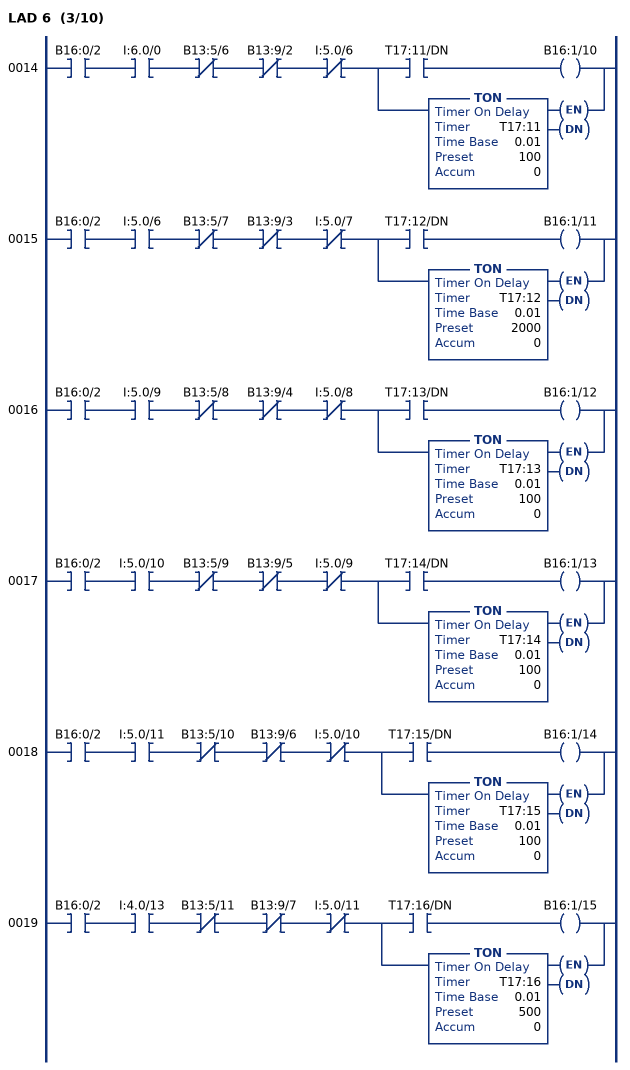
% Rung: 14 %
SOR XIC B16:0/2 XIC I:6.0/0 XIO B13:5/6 XIO B13:9/2 XIO I:5.0/6 BST XIC T17:11/DN OTE B16:1/10 NXB TON T17:11 0.01 100 0 BND EOR
% Rung: 15 %
SOR XIC B16:0/2 XIC I:5.0/6 XIO B13:5/7 XIO B13:9/3 XIO I:5.0/7 BST XIC T17:12/DN OTE B16:1/11 NXB TON T17:12 0.01 2000 0 BND EOR
% Rung: 16 %
SOR XIC B16:0/2 XIC I:5.0/9 XIO B13:5/8 XIO B13:9/4 XIO I:5.0/8 BST XIC T17:13/DN OTE B16:1/12 NXB TON T17:13 0.01 100 0 BND EOR
% Rung: 17 %
SOR XIC B16:0/2 XIC I:5.0/10 XIO B13:5/9 XIO B13:9/5 XIO I:5.0/9 BST XIC T17:14/DN OTE B16:1/13 NXB TON T17:14 0.01 100 0 BND EOR
% Rung: 18 %
SOR XIC B16:0/2 XIC I:5.0/11 XIO B13:5/10 XIO B13:9/6 XIO I:5.0/10 BST XIC T17:15/DN OTE B16:1/14 NXB TON T17:15 0.01 100 0 BND EOR
% Rung: 19 %
SOR XIC B16:0/2 XIC I:4.0/13 XIO B13:5/11 XIO B13:9/7 XIO I:5.0/11 BST XIC T17:16/DN OTE B16:1/15 NXB TON T17:16 0.01 500 0 BND EOR

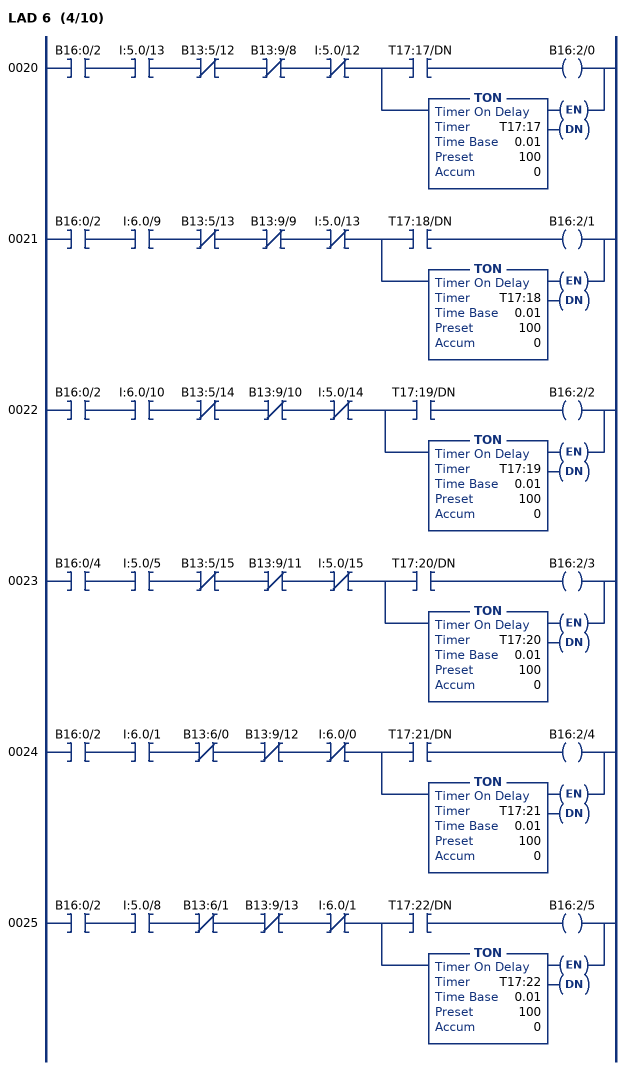
% Rung: 20 %
SOR XIC B16:0/2 XIC I:5.0/13 XIO B13:5/12 XIO B13:9/8 XIO I:5.0/12 BST XIC T17:17/DN OTE B16:2/0 NXB TON T17:17 0.01 100 0 BND EOR
% Rung: 21 %
SOR XIC B16:0/2 XIC I:6.0/9 XIO B13:5/13 XIO B13:9/9 XIO I:5.0/13 BST XIC T17:18/DN OTE B16:2/1 NXB TON T17:18 0.01 100 0 BND EOR
% Rung: 22 %
SOR XIC B16:0/2 XIC I:6.0/10 XIO B13:5/14 XIO B13:9/10 XIO I:5.0/14 BST XIC T17:19/DN OTE B16:2/2 NXB TON T17:19 0.01 100 0 BND EOR
% Rung: 23 %
SOR XIC B16:0/4 XIC I:5.0/5 XIO B13:5/15 XIO B13:9/11 XIO I:5.0/15 BST XIC T17:20/DN OTE B16:2/3 NXB TON T17:20 0.01 100 0 BND EOR
% Rung: 24 %
SOR XIC B16:0/2 XIC I:6.0/1 XIO B13:6/0 XIO B13:9/12 XIO I:6.0/0 BST XIC T17:21/DN OTE B16:2/4 NXB TON T17:21 0.01 100 0 BND EOR
% Rung: 25 %
SOR XIC B16:0/2 XIC I:5.0/8 XIO B13:6/1 XIO B13:9/13 XIO I:6.0/1 BST XIC T17:22/DN OTE B16:2/5 NXB TON T17:22 0.01 100 0 BND EOR

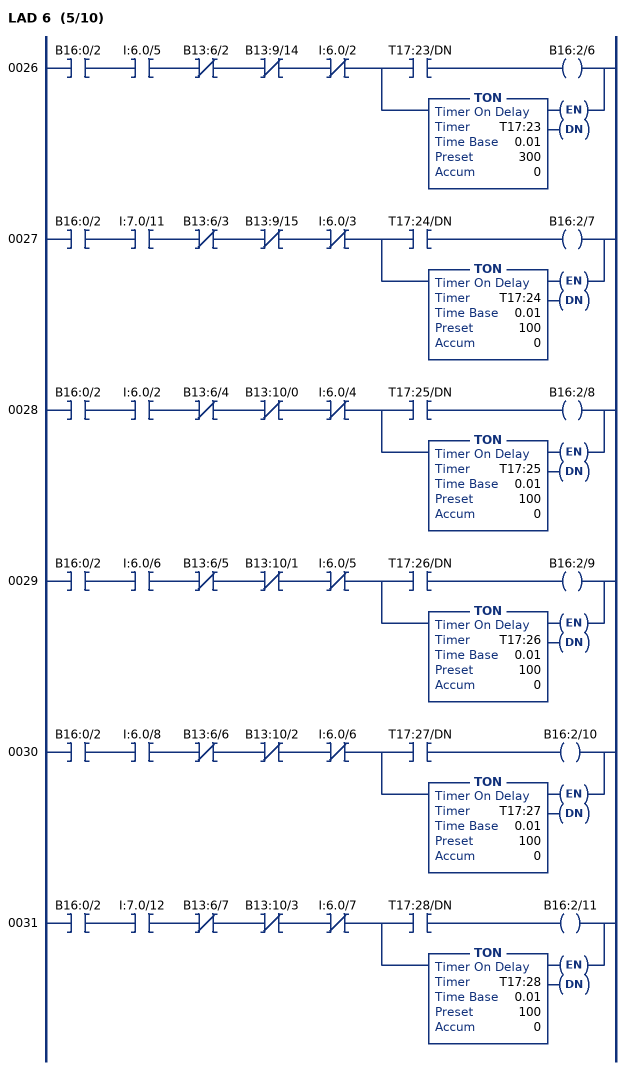
% Rung: 26 %
SOR XIC B16:0/2 XIC I:6.0/5 XIO B13:6/2 XIO B13:9/14 XIO I:6.0/2 BST XIC T17:23/DN OTE B16:2/6 NXB TON T17:23 0.01 300 0 BND EOR
% Rung: 27 %
SOR XIC B16:0/2 XIC I:7.0/11 XIO B13:6/3 XIO B13:9/15 XIO I:6.0/3 BST XIC T17:24/DN OTE B16:2/7 NXB TON T17:24 0.01 100 0 BND EOR
% Rung: 28 %
SOR XIC B16:0/2 XIC I:6.0/2 XIO B13:6/4 XIO B13:10/0 XIO I:6.0/4 BST XIC T17:25/DN OTE B16:2/8 NXB TON T17:25 0.01 100 0 BND EOR
% Rung: 29 %
SOR XIC B16:0/2 XIC I:6.0/6 XIO B13:6/5 XIO B13:10/1 XIO I:6.0/5 BST XIC T17:26/DN OTE B16:2/9 NXB TON T17:26 0.01 100 0 BND EOR
% Rung: 30 %
SOR XIC B16:0/2 XIC I:6.0/8 XIO B13:6/6 XIO B13:10/2 XIO I:6.0/6 BST XIC T17:27/DN OTE B16:2/10 NXB TON T17:27 0.01 100 0 BND EOR
% Rung: 31 %
SOR XIC B16:0/2 XIC I:7.0/12 XIO B13:6/7 XIO B13:10/3 XIO I:6.0/7 BST XIC T17:28/DN OTE B16:2/11 NXB TON T17:28 0.01 100 0 BND EOR

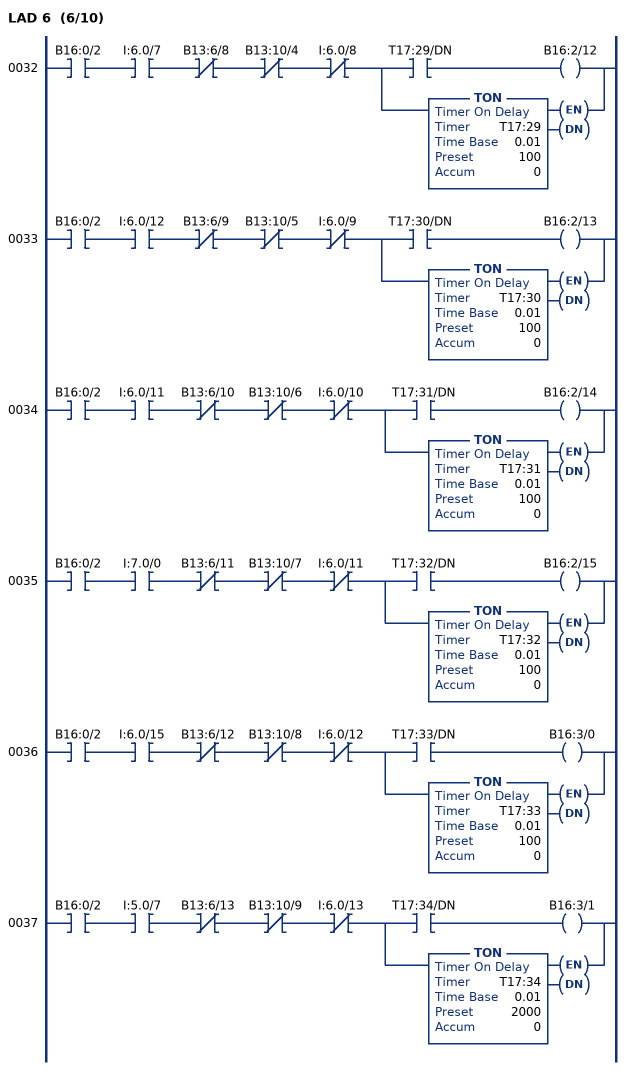
% Rung: 32 %
SOR XIC B16:0/2 XIC I:6.0/7 XIO B13:6/8 XIO B13:10/4 XIO I:6.0/8 BST XIC T17:29/DN OTE B16:2/12 NXB TON T17:29 0.01 100 0 BND EOR
% Rung: 33 %
SOR XIC B16:0/2 XIC I:6.0/12 XIO B13:6/9 XIO B13:10/5 XIO I:6.0/9 BST XIC T17:30/DN OTE B16:2/13 NXB TON T17:30 0.01 100 0 BND EOR
% Rung: 34 %
SOR XIC B16:0/2 XIC I:6.0/11 XIO B13:6/10 XIO B13:10/6 XIO I:6.0/10 BST XIC T17:31/DN OTE B16:2/14 NXB TON T17:31 0.01 100 0 BND EOR
% Rung: 35 %
SOR XIC B16:0/2 XIC I:7.0/0 XIO B13:6/11 XIO B13:10/7 XIO I:6.0/11 BST XIC T17:32/DN OTE B16:2/15 NXB TON T17:32 0.01 100 0 BND EOR
% Rung: 36 %
SOR XIC B16:0/2 XIC I:6.0/15 XIO B13:6/12 XIO B13:10/8 XIO I:6.0/12 BST XIC T17:33/DN OTE B16:3/0 NXB TON T17:33 0.01 100 0 BND EOR
% Rung: 37 %
SOR XIC B16:0/2 XIC I:5.0/7 XIO B13:6/13 XIO B13:10/9 XIO I:6.0/13 BST XIC T17:34/DN OTE B16:3/1 NXB TON T17:34 0.01 2000 0 BND EOR

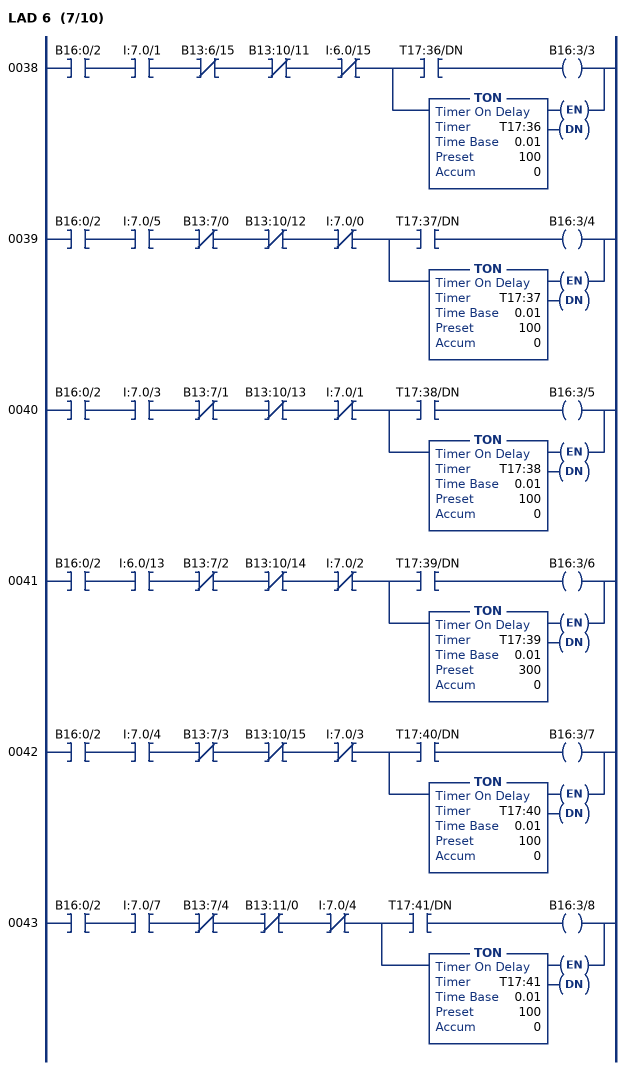
% Rung: 38 %
SOR XIC B16:0/2 XIC I:7.0/1 XIO B13:6/15 XIO B13:10/11 XIO I:6.0/15 BST XIC T17:36/DN OTE B16:3/3 NXB TON T17:36 0.01 100 0 BND EOR
% Rung: 39 %
SOR XIC B16:0/2 XIC I:7.0/5 XIO B13:7/0 XIO B13:10/12 XIO I:7.0/0 BST XIC T17:37/DN OTE B16:3/4 NXB TON T17:37 0.01 100 0 BND EOR
% Rung: 40 %
SOR XIC B16:0/2 XIC I:7.0/3 XIO B13:7/1 XIO B13:10/13 XIO I:7.0/1 BST XIC T17:38/DN OTE B16:3/5 NXB TON T17:38 0.01 100 0 BND EOR
% Rung: 41 %
SOR XIC B16:0/2 XIC I:6.0/13 XIO B13:7/2 XIO B13:10/14 XIO I:7.0/2 BST XIC T17:39/DN OTE B16:3/6 NXB TON T17:39 0.01 300 0 BND EOR
% Rung: 42 %
SOR XIC B16:0/2 XIC I:7.0/4 XIO B13:7/3 XIO B13:10/15 XIO I:7.0/3 BST XIC T17:40/DN OTE B16:3/7 NXB TON T17:40 0.01 100 0 BND EOR
% Rung: 43 %
SOR XIC B16:0/2 XIC I:7.0/7 XIO B13:7/4 XIO B13:11/0 XIO I:7.0/4 BST XIC T17:41/DN OTE B16:3/8 NXB TON T17:41 0.01 100 0 BND EOR

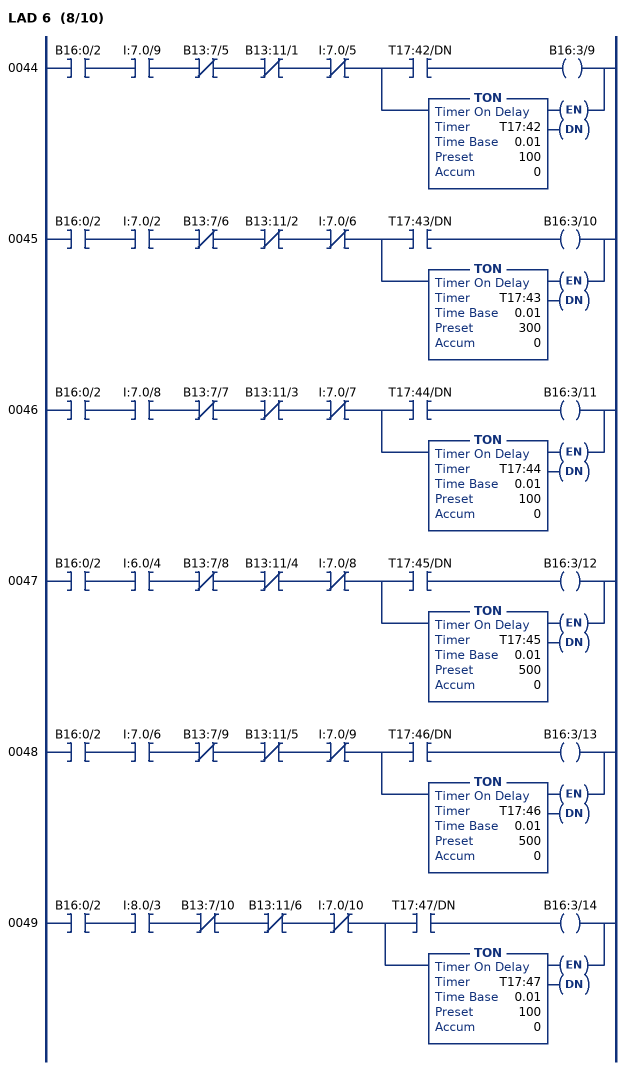
% Rung: 44 %
SOR XIC B16:0/2 XIC I:7.0/9 XIO B13:7/5 XIO B13:11/1 XIO I:7.0/5 BST XIC T17:42/DN OTE B16:3/9 NXB TON T17:42 0.01 100 0 BND EOR
% Rung: 45 %
SOR XIC B16:0/2 XIC I:7.0/2 XIO B13:7/6 XIO B13:11/2 XIO I:7.0/6 BST XIC T17:43/DN OTE B16:3/10 NXB TON T17:43 0.01 300 0 BND EOR
% Rung: 46 %
SOR XIC B16:0/2 XIC I:7.0/8 XIO B13:7/7 XIO B13:11/3 XIO I:7.0/7 BST XIC T17:44/DN OTE B16:3/11 NXB TON T17:44 0.01 100 0 BND EOR
% Rung: 47 %
SOR XIC B16:0/2 XIC I:6.0/4 XIO B13:7/8 XIO B13:11/4 XIO I:7.0/8 BST XIC T17:45/DN OTE B16:3/12 NXB TON T17:45 0.01 500 0 BND EOR
% Rung: 48 %
SOR XIC B16:0/2 XIC I:7.0/6 XIO B13:7/9 XIO B13:11/5 XIO I:7.0/9 BST XIC T17:46/DN OTE B16:3/13 NXB TON T17:46 0.01 500 0 BND EOR
% Rung: 49 %
SOR XIC B16:0/2 XIC I:8.0/3 XIO B13:7/10 XIO B13:11/6 XIO I:7.0/10 BST XIC T17:47/DN OTE B16:3/14 NXB TON T17:47 0.01 100 0 BND EOR

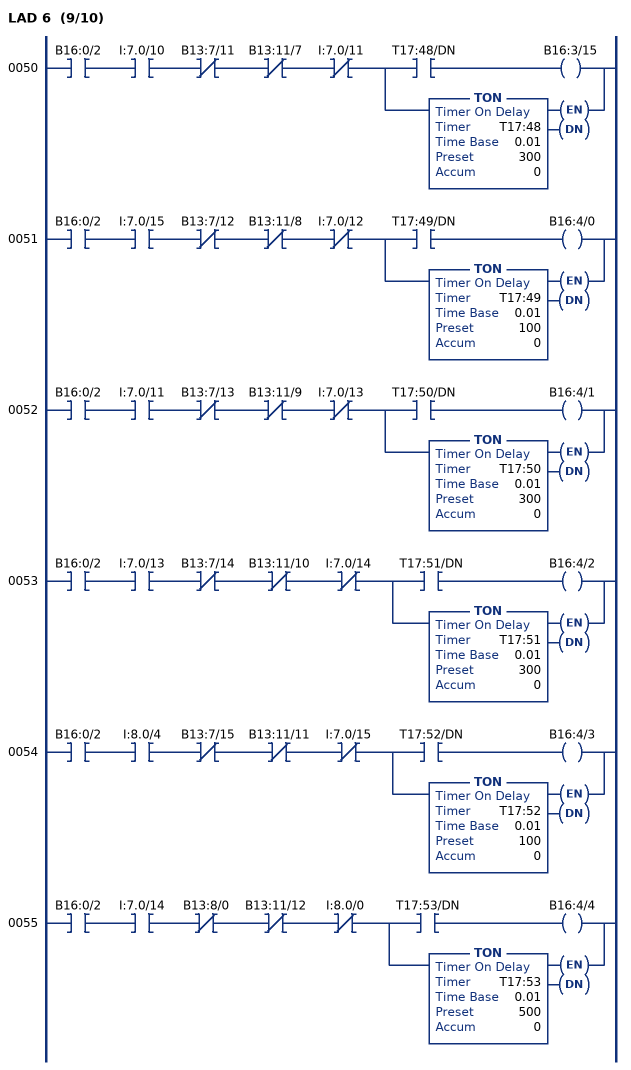
% Rung: 50 %
SOR XIC B16:0/2 XIC I:7.0/10 XIO B13:7/11 XIO B13:11/7 XIO I:7.0/11 BST XIC T17:48/DN OTE B16:3/15 NXB TON T17:48 0.01 300 0 BND EOR
% Rung: 51 %
SOR XIC B16:0/2 XIC I:7.0/15 XIO B13:7/12 XIO B13:11/8 XIO I:7.0/12 BST XIC T17:49/DN OTE B16:4/0 NXB TON T17:49 0.01 100 0 BND EOR
% Rung: 52 %
SOR XIC B16:0/2 XIC I:7.0/11 XIO B13:7/13 XIO B13:11/9 XIO I:7.0/13 BST XIC T17:50/DN OTE B16:4/1 NXB TON T17:50 0.01 300 0 BND EOR
% Rung: 53 %
SOR XIC B16:0/2 XIC I:7.0/13 XIO B13:7/14 XIO B13:11/10 XIO I:7.0/14 BST XIC T17:51/DN OTE B16:4/2 NXB TON T17:51 0.01 300 0 BND EOR
% Rung: 54 %
SOR XIC B16:0/2 XIC I:8.0/4 XIO B13:7/15 XIO B13:11/11 XIO I:7.0/15 BST XIC T17:52/DN OTE B16:4/3 NXB TON T17:52 0.01 100 0 BND EOR
% Rung: 55 %
SOR XIC B16:0/2 XIC I:7.0/14 XIO B13:8/0 XIO B13:11/12 XIO I:8.0/0 BST XIC T17:53/DN OTE B16:4/4 NXB TON T17:53 0.01 500 0 BND EOR

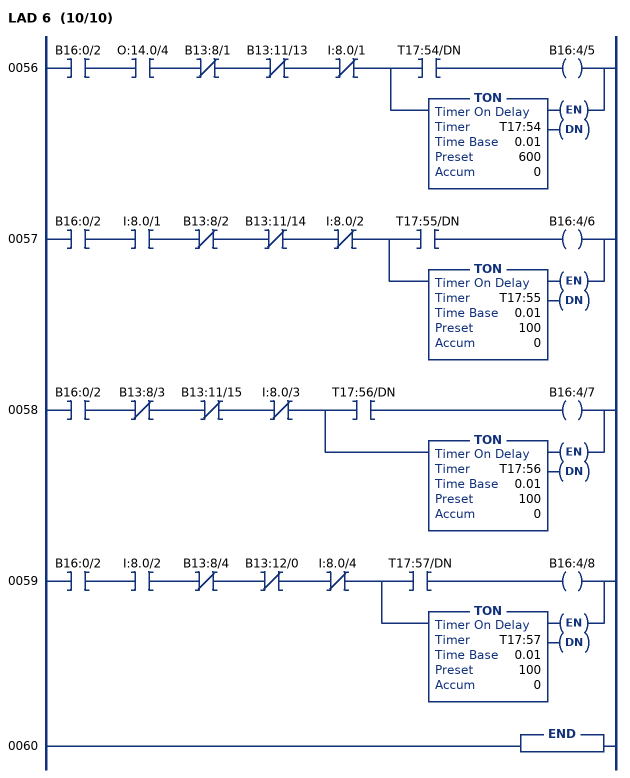
% Rung: 56 %
SOR XIC B16:0/2 XIC O:14.0/4 XIO B13:8/1 XIO B13:11/13 XIO I:8.0/1 BST XIC T17:54/DN OTE B16:4/5 NXB TON T17:54 0.01 600 0 BND EOR
% Rung: 57 %
SOR XIC B16:0/2 XIC I:8.0/1 XIO B13:8/2 XIO B13:11/14 XIO I:8.0/2 BST XIC T17:55/DN OTE B16:4/6 NXB TON T17:55 0.01 100 0 BND EOR
% Rung: 58 %
SOR XIC B16:0/2 XIO B13:8/3 XIO B13:11/15 XIO I:8.0/3 BST XIC T17:56/DN OTE B16:4/7 NXB TON T17:56 0.01 100 0 BND EOR
% Rung: 59 %
SOR XIC B16:0/2 XIC I:8.0/2 XIO B13:8/4 XIO B13:12/0 XIO I:8.0/4 BST XIC T17:57/DN OTE B16:4/8 NXB TON T17:57 0.01 100 0 BND EOR
% Rung: 60 %
SOR END EOR

LADDER 7
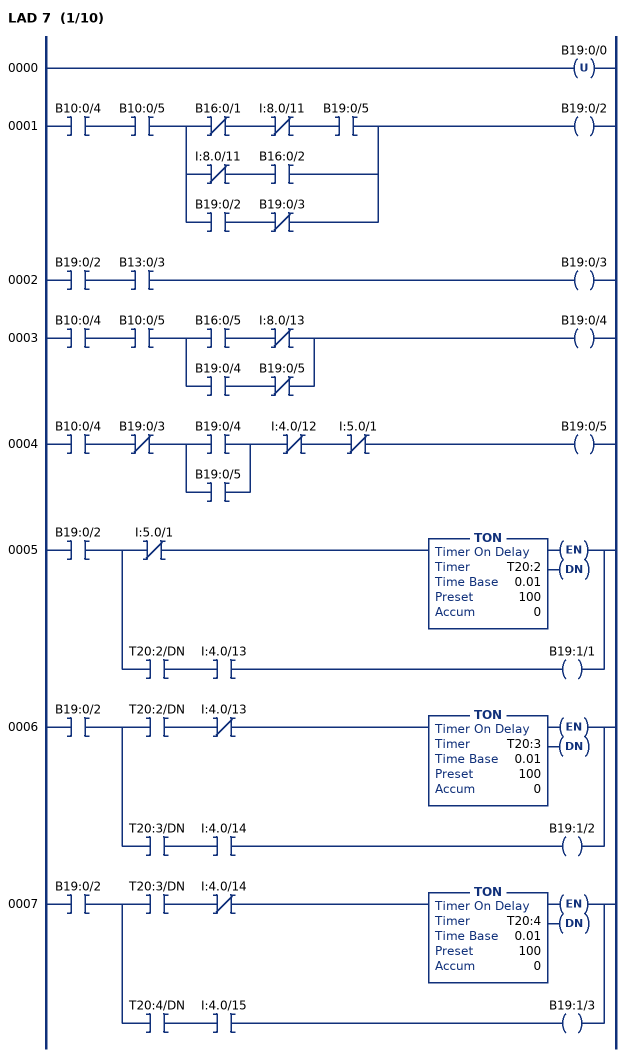
% Rung: 0 %
SOR OTU B19:0/0 EOR
% Rung: 1 %
SOR XIC B10:0/4 XIC B10:0/5 BST XIO B16:0/1 XIO I:8.0/11 XIC B19:0/5 NXB XIO I:8.0/11 XIC B16:0/2 NXB XIC B19:0/2 XIO B19:0/3 BND OTE B19:0/2 EOR
% Rung: 2 %
SOR XIC B19:0/2 XIC B13:0/3 OTE B19:0/3 EOR
% Rung: 3 %
SOR XIC B10:0/4 XIC B10:0/5 BST XIC B16:0/5 XIO I:8.0/13 NXB XIC B19:0/4 XIO B19:0/5 BND OTE B19:0/4 EOR
% Rung: 4 %
SOR XIC B10:0/4 XIO B19:0/3 BST XIC B19:0/4 NXB XIC B19:0/5 BND XIO I:4.0/12 XIO I:5.0/1 OTE B19:0/5 EOR
% Rung: 5 %
SOR XIC B19:0/2 BST XIO I:5.0/1 TON T20:2 0.01 100 0 NXB XIC T20:2/DN XIC I:4.0/13 OTE B19:1/1 BND EOR
% Rung: 6 %
SOR XIC B19:0/2 BST XIC T20:2/DN XIO I:4.0/13 TON T20:3 0.01 100 0 NXB XIC T20:3/DN XIC I:4.0/14 OTE B19:1/2 BND EOR
% Rung: 7 %
SOR XIC B19:0/2 BST XIC T20:3/DN XIO I:4.0/14 TON T20:4 0.01 100 0 NXB XIC T20:4/DN XIC I:4.0/15 OTE B19:1/3 BND EOR

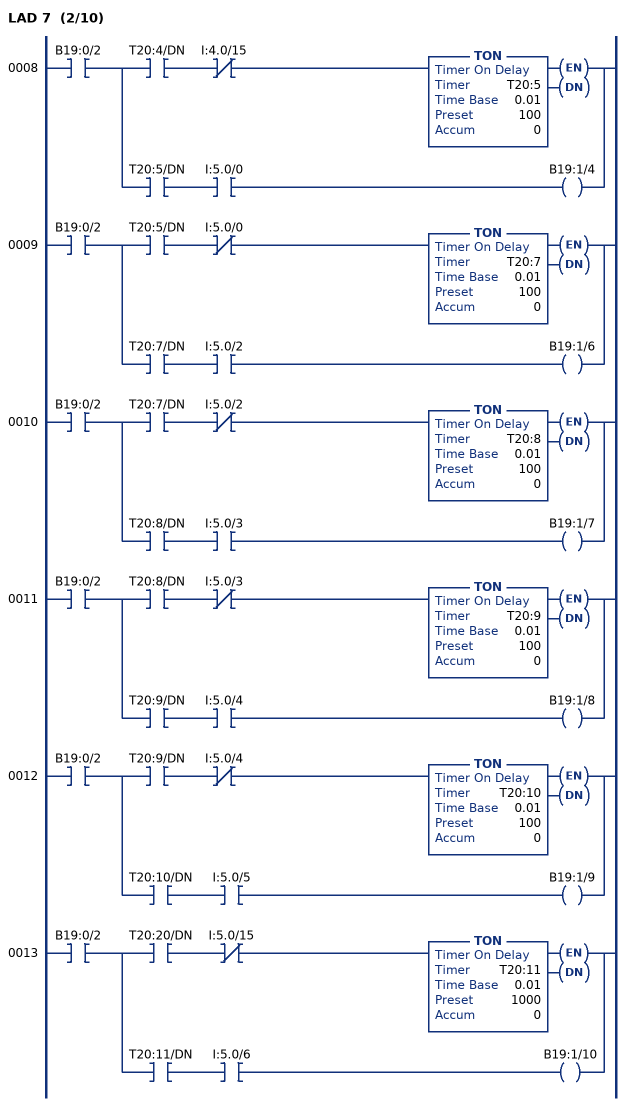
% Rung: 8 %
SOR XIC B19:0/2 BST XIC T20:4/DN XIO I:4.0/15 TON T20:5 0.01 100 0 NXB XIC T20:5/DN XIC I:5.0/0 OTE B19:1/4 BND EOR
% Rung: 9 %
SOR XIC B19:0/2 BST XIC T20:5/DN XIO I:5.0/0 TON T20:7 0.01 100 0 NXB XIC T20:7/DN XIC I:5.0/2 OTE B19:1/6 BND EOR
% Rung: 10 %
SOR XIC B19:0/2 BST XIC T20:7/DN XIO I:5.0/2 TON T20:8 0.01 100 0 NXB XIC T20:8/DN XIC I:5.0/3 OTE B19:1/7 BND EOR
% Rung: 11 %
SOR XIC B19:0/2 BST XIC T20:8/DN XIO I:5.0/3 TON T20:9 0.01 100 0 NXB XIC T20:9/DN XIC I:5.0/4 OTE B19:1/8 BND EOR
% Rung: 12 %
SOR XIC B19:0/2 BST XIC T20:9/DN XIO I:5.0/4 TON T20:10 0.01 100 0 NXB XIC T20:10/DN XIC I:5.0/5 OTE B19:1/9 BND EOR
% Rung: 13 %
SOR XIC B19:0/2 BST XIC T20:20/DN XIO I:5.0/15 TON T20:11 0.01 1000 0 NXB XIC T20:11/DN XIC I:5.0/6 OTE B19:1/10 BND EOR

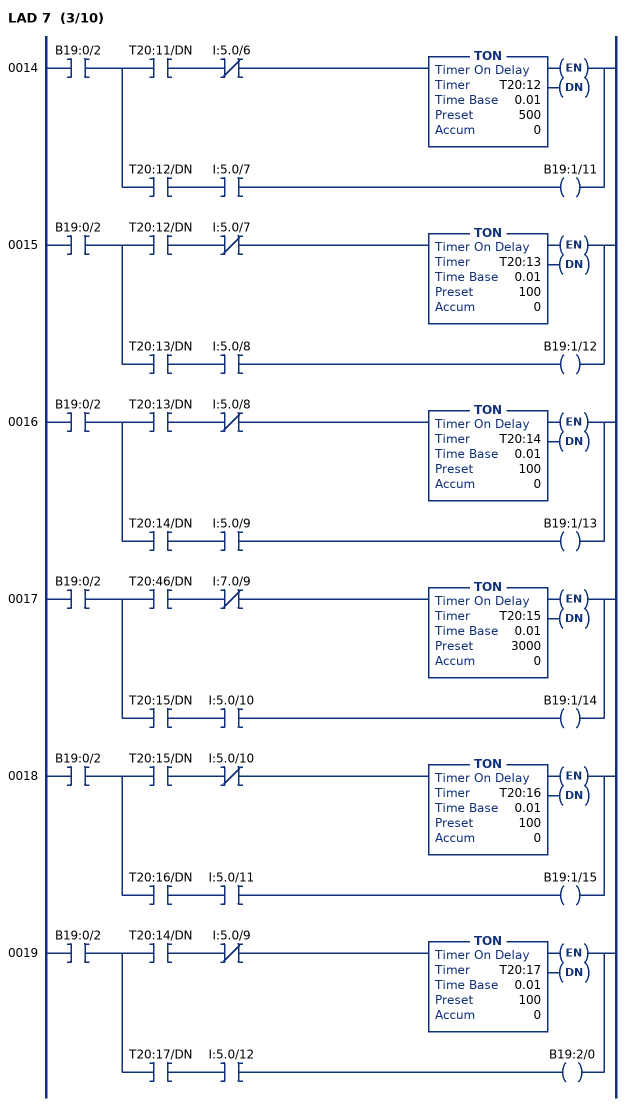
% Rung: 14 %
SOR XIC B19:0/2 BST XIC T20:11/DN XIO I:5.0/6 TON T20:12 0.01 500 0 NXB XIC T20:12/DN XIC I:5.0/7 OTE B19:1/11 BND EOR
% Rung: 15 %
SOR XIC B19:0/2 BST XIC T20:12/DN XIO I:5.0/7 TON T20:13 0.01 100 0 NXB XIC T20:13/DN XIC I:5.0/8 OTE B19:1/12 BND EOR
% Rung: 16 %
SOR XIC B19:0/2 BST XIC T20:13/DN XIO I:5.0/8 TON T20:14 0.01 100 0 NXB XIC T20:14/DN XIC I:5.0/9 OTE B19:1/13 BND EOR
% Rung: 17 %
SOR XIC B19:0/2 BST XIC T20:46/DN XIO I:7.0/9 TON T20:15 0.01 3000 0 NXB XIC T20:15/DN XIC I:5.0/10 OTE B19:1/14 BND EOR
% Rung: 18 %
SOR XIC B19:0/2 BST XIC T20:15/DN XIO I:5.0/10 TON T20:16 0.01 100 0 NXB XIC T20:16/DN XIC I:5.0/11 OTE B19:1/15 BND EOR
% Rung: 19 %
SOR XIC B19:0/2 BST XIC T20:14/DN XIO I:5.0/9 TON T20:17 0.01 100 0 NXB XIC T20:17/DN XIC I:5.0/12 OTE B19:2/0 BND EOR

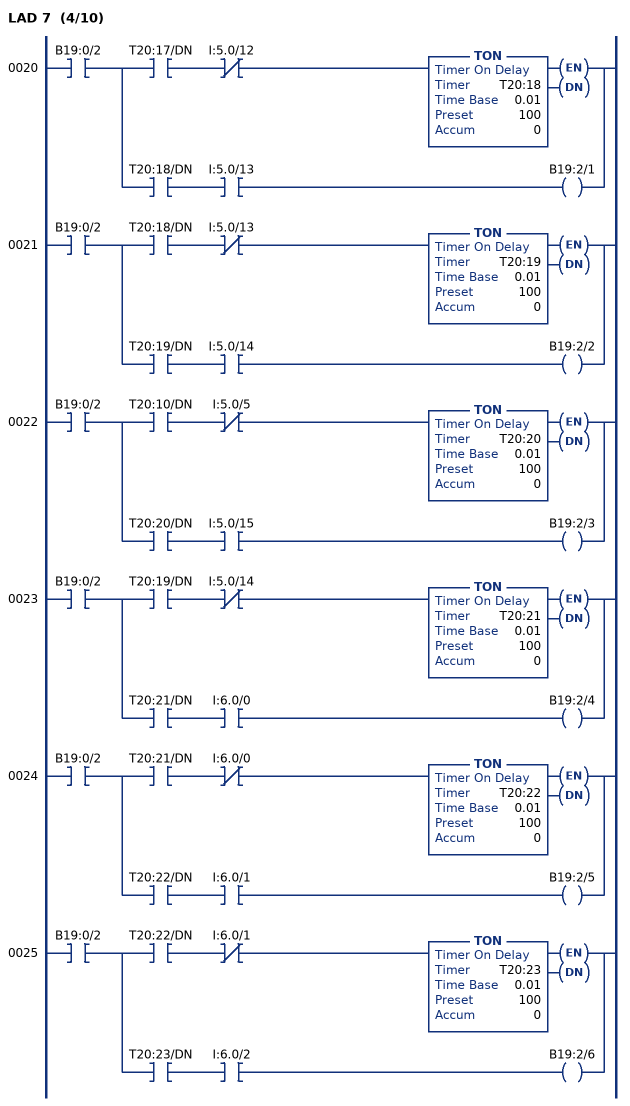
% Rung: 20 %
SOR XIC B19:0/2 BST XIC T20:17/DN XIO I:5.0/12 TON T20:18 0.01 100 0 NXB XIC T20:18/DN XIC I:5.0/13 OTE B19:2/1 BND EOR
% Rung: 21 %
SOR XIC B19:0/2 BST XIC T20:18/DN XIO I:5.0/13 TON T20:19 0.01 100 0 NXB XIC T20:19/DN XIC I:5.0/14 OTE B19:2/2 BND EOR
% Rung: 22 %
SOR XIC B19:0/2 BST XIC T20:10/DN XIO I:5.0/5 TON T20:20 0.01 100 0 NXB XIC T20:20/DN XIC I:5.0/15 OTE B19:2/3 BND EOR
% Rung: 23 %
SOR XIC B19:0/2 BST XIC T20:19/DN XIO I:5.0/14 TON T20:21 0.01 100 0 NXB XIC T20:21/DN XIC I:6.0/0 OTE B19:2/4 BND EOR
% Rung: 24 %
SOR XIC B19:0/2 BST XIC T20:21/DN XIO I:6.0/0 TON T20:22 0.01 100 0 NXB XIC T20:22/DN XIC I:6.0/1 OTE B19:2/5 BND EOR
% Rung: 25 %
SOR XIC B19:0/2 BST XIC T20:22/DN XIO I:6.0/1 TON T20:23 0.01 100 0 NXB XIC T20:23/DN XIC I:6.0/2 OTE B19:2/6 BND EOR

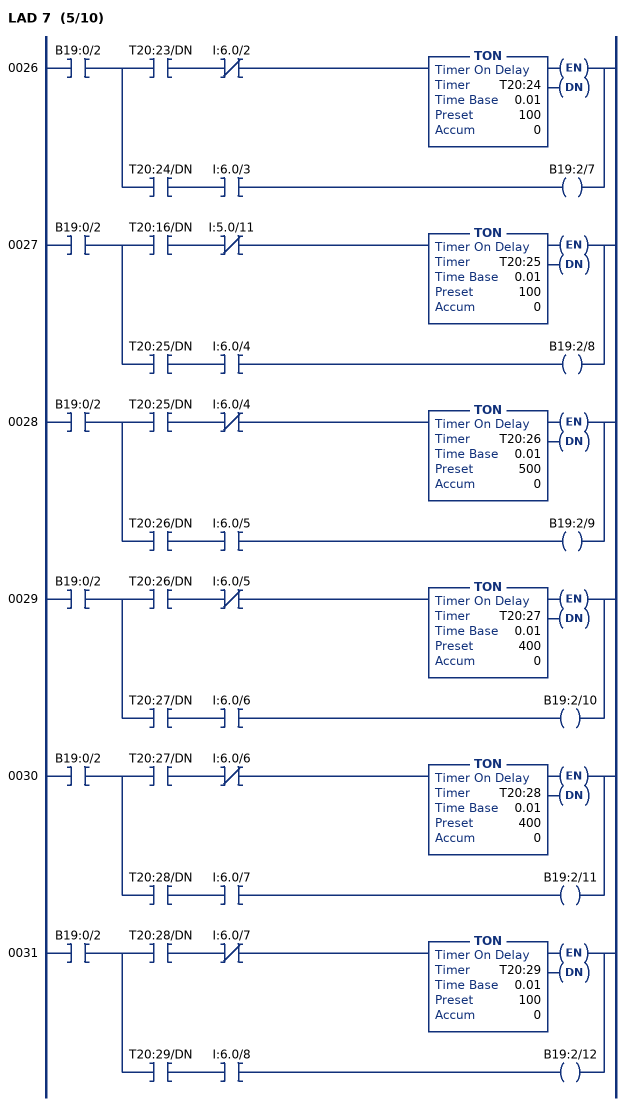
% Rung: 26 %
SOR XIC B19:0/2 BST XIC T20:23/DN XIO I:6.0/2 TON T20:24 0.01 100 0 NXB XIC T20:24/DN XIC I:6.0/3 OTE B19:2/7 BND EOR
% Rung: 27 %
SOR XIC B19:0/2 BST XIC T20:16/DN XIO I:5.0/11 TON T20:25 0.01 100 0 NXB XIC T20:25/DN XIC I:6.0/4 OTE B19:2/8 BND EOR
% Rung: 28 %
SOR XIC B19:0/2 BST XIC T20:25/DN XIO I:6.0/4 TON T20:26 0.01 500 0 NXB XIC T20:26/DN XIC I:6.0/5 OTE B19:2/9 BND EOR
% Rung: 29 %
SOR XIC B19:0/2 BST XIC T20:26/DN XIO I:6.0/5 TON T20:27 0.01 400 0 NXB XIC T20:27/DN XIC I:6.0/6 OTE B19:2/10 BND EOR
% Rung: 30 %
SOR XIC B19:0/2 BST XIC T20:27/DN XIO I:6.0/6 TON T20:28 0.01 400 0 NXB XIC T20:28/DN XIC I:6.0/7 OTE B19:2/11 BND EOR
% Rung: 31 %
SOR XIC B19:0/2 BST XIC T20:28/DN XIO I:6.0/7 TON T20:29 0.01 100 0 NXB XIC T20:29/DN XIC I:6.0/8 OTE B19:2/12 BND EOR

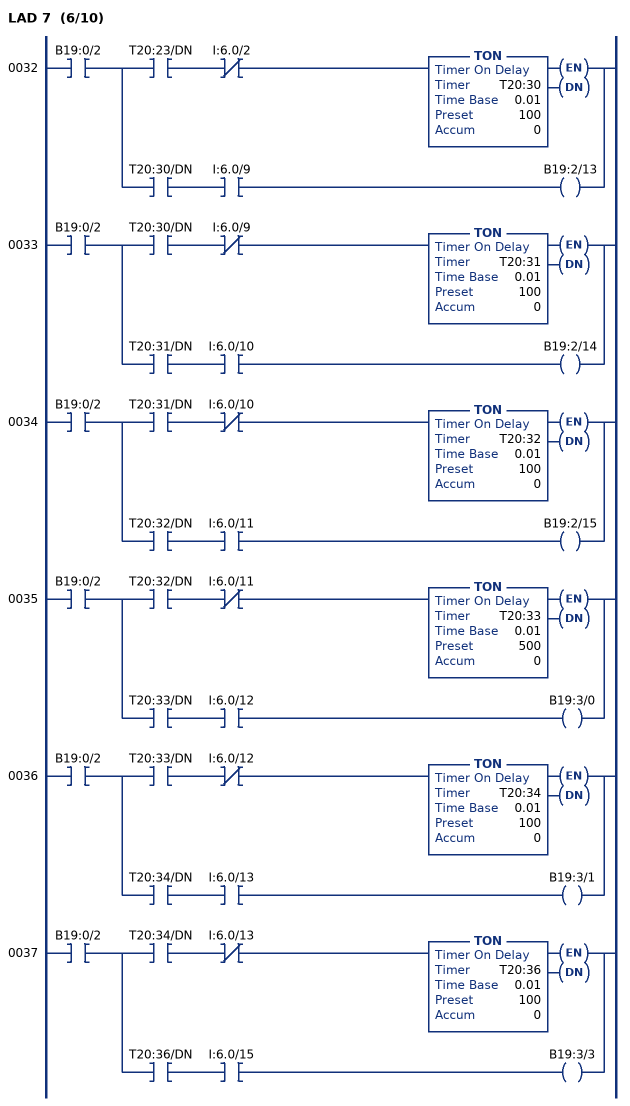
% Rung: 32 %
SOR XIC B19:0/2 BST XIC T20:23/DN XIO I:6.0/2 TON T20:30 0.01 100 0 NXB XIC T20:30/DN XIC I:6.0/9 OTE B19:2/13 BND EOR
% Rung: 33 %
SOR XIC B19:0/2 BST XIC T20:30/DN XIO I:6.0/9 TON T20:31 0.01 100 0 NXB XIC T20:31/DN XIC I:6.0/10 OTE B19:2/14 BND EOR
% Rung: 34 %
SOR XIC B19:0/2 BST XIC T20:31/DN XIO I:6.0/10 TON T20:32 0.01 100 0 NXB XIC T20:32/DN XIC I:6.0/11 OTE B19:2/15 BND EOR
% Rung: 35 %
SOR XIC B19:0/2 BST XIC T20:32/DN XIO I:6.0/11 TON T20:33 0.01 500 0 NXB XIC T20:33/DN XIC I:6.0/12 OTE B19:3/0 BND EOR
% Rung: 36 %
SOR XIC B19:0/2 BST XIC T20:33/DN XIO I:6.0/12 TON T20:34 0.01 100 0 NXB XIC T20:34/DN XIC I:6.0/13 OTE B19:3/1 BND EOR
% Rung: 37 %
SOR XIC B19:0/2 BST XIC T20:34/DN XIO I:6.0/13 TON T20:36 0.01 100 0 NXB XIC T20:36/DN XIC I:6.0/15 OTE B19:3/3 BND EOR

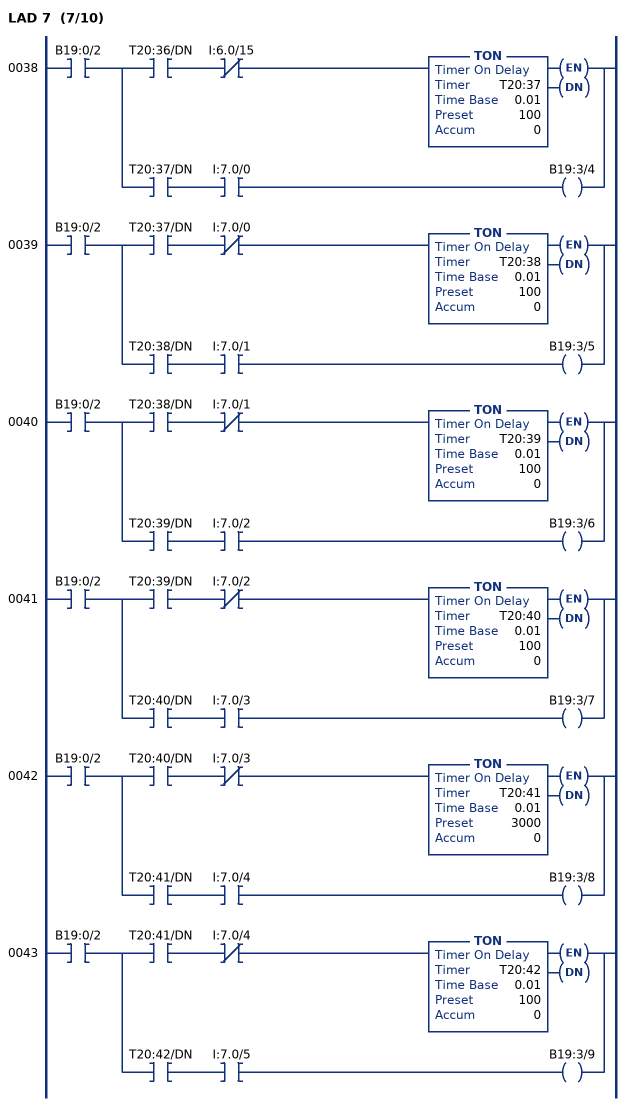
% Rung: 38 %
SOR XIC B19:0/2 BST XIC T20:36/DN XIO I:6.0/15 TON T20:37 0.01 100 0 NXB XIC T20:37/DN XIC I:7.0/0 OTE B19:3/4 BND EOR
% Rung: 39 %
SOR XIC B19:0/2 BST XIC T20:37/DN XIO I:7.0/0 TON T20:38 0.01 100 0 NXB XIC T20:38/DN XIC I:7.0/1 OTE B19:3/5 BND EOR
% Rung: 40 %
SOR XIC B19:0/2 BST XIC T20:38/DN XIO I:7.0/1 TON T20:39 0.01 100 0 NXB XIC T20:39/DN XIC I:7.0/2 OTE B19:3/6 BND EOR
% Rung: 41 %
SOR XIC B19:0/2 BST XIC T20:39/DN XIO I:7.0/2 TON T20:40 0.01 100 0 NXB XIC T20:40/DN XIC I:7.0/3 OTE B19:3/7 BND EOR
% Rung: 42 %
SOR XIC B19:0/2 BST XIC T20:40/DN XIO I:7.0/3 TON T20:41 0.01 3000 0 NXB XIC T20:41/DN XIC I:7.0/4 OTE B19:3/8 BND EOR
% Rung: 43 %
SOR XIC B19:0/2 BST XIC T20:41/DN XIO I:7.0/4 TON T20:42 0.01 100 0 NXB XIC T20:42/DN XIC I:7.0/5 OTE B19:3/9 BND EOR

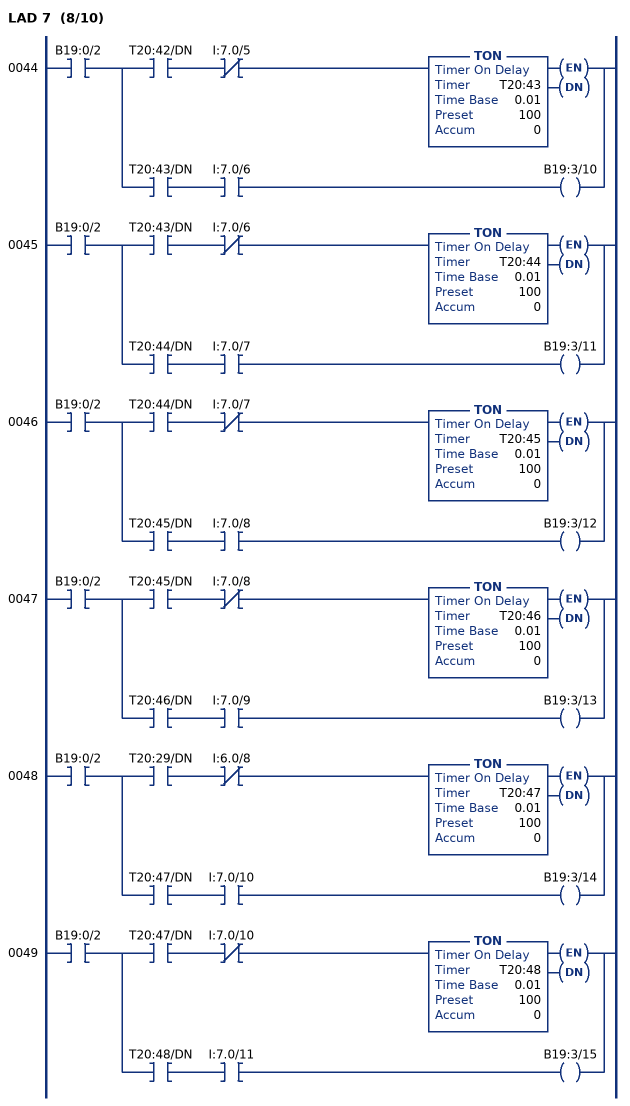
% Rung: 44 %
SOR XIC B19:0/2 BST XIC T20:42/DN XIO I:7.0/5 TON T20:43 0.01 100 0 NXB XIC T20:43/DN XIC I:7.0/6 OTE B19:3/10 BND EOR
% Rung: 45 %
SOR XIC B19:0/2 BST XIC T20:43/DN XIO I:7.0/6 TON T20:44 0.01 100 0 NXB XIC T20:44/DN XIC I:7.0/7 OTE B19:3/11 BND EOR
% Rung: 46 %
SOR XIC B19:0/2 BST XIC T20:44/DN XIO I:7.0/7 TON T20:45 0.01 100 0 NXB XIC T20:45/DN XIC I:7.0/8 OTE B19:3/12 BND EOR
% Rung: 47 %
SOR XIC B19:0/2 BST XIC T20:45/DN XIO I:7.0/8 TON T20:46 0.01 100 0 NXB XIC T20:46/DN XIC I:7.0/9 OTE B19:3/13 BND EOR
% Rung: 48 %
SOR XIC B19:0/2 BST XIC T20:29/DN XIO I:6.0/8 TON T20:47 0.01 100 0 NXB XIC T20:47/DN XIC I:7.0/10 OTE B19:3/14 BND EOR
% Rung: 49 %
SOR XIC B19:0/2 BST XIC T20:47/DN XIO I:7.0/10 TON T20:48 0.01 100 0 NXB XIC T20:48/DN XIC I:7.0/11 OTE B19:3/15 BND EOR

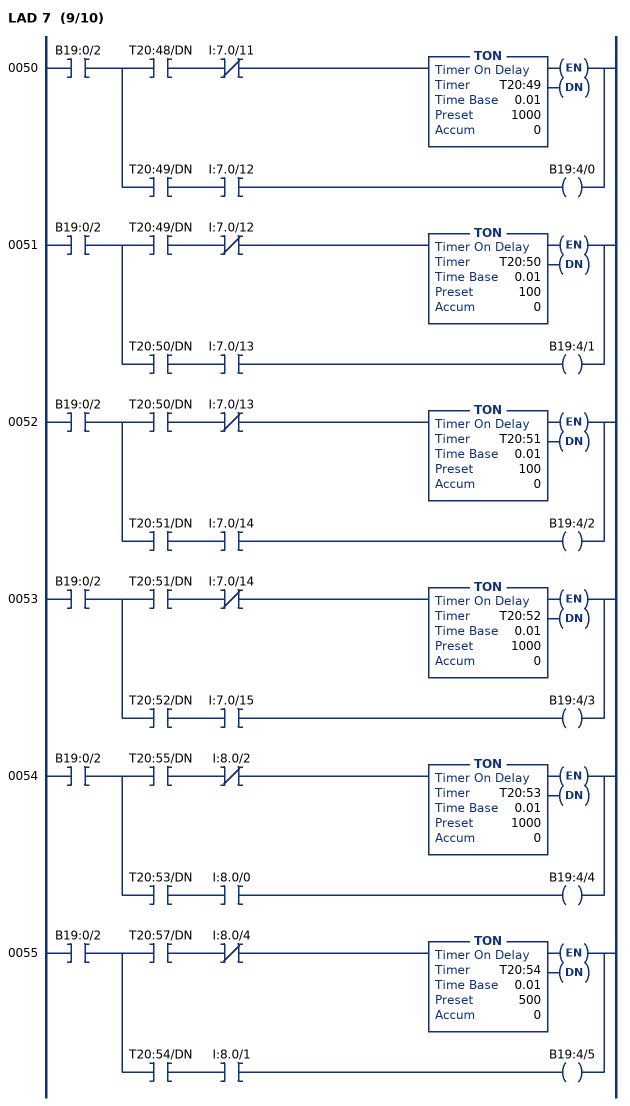
% Rung: 50 %
SOR XIC B19:0/2 BST XIC T20:48/DN XIO I:7.0/11 TON T20:49 0.01 1000 0 NXB XIC T20:49/DN XIC I:7.0/12 OTE B19:4/0 BND EOR
% Rung: 51 %
SOR XIC B19:0/2 BST XIC T20:49/DN XIO I:7.0/12 TON T20:50 0.01 100 0 NXB XIC T20:50/DN XIC I:7.0/13 OTE B19:4/1 BND EOR
% Rung: 52 %
SOR XIC B19:0/2 BST XIC T20:50/DN XIO I:7.0/13 TON T20:51 0.01 100 0 NXB XIC T20:51/DN XIC I:7.0/14 OTE B19:4/2 BND EOR
% Rung: 53 %
SOR XIC B19:0/2 BST XIC T20:51/DN XIO I:7.0/14 TON T20:52 0.01 1000 0 NXB XIC T20:52/DN XIC I:7.0/15 OTE B19:4/3 BND EOR
% Rung: 54 %
SOR XIC B19:0/2 BST XIC T20:55/DN XIO I:8.0/2 TON T20:53 0.01 1000 0 NXB XIC T20:53/DN XIC I:8.0/0 OTE B19:4/4 BND EOR
% Rung: 55 %
SOR XIC B19:0/2 BST XIC T20:57/DN XIO I:8.0/4 TON T20:54 0.01 500 0 NXB XIC T20:54/DN XIC I:8.0/1 OTE B19:4/5 BND EOR

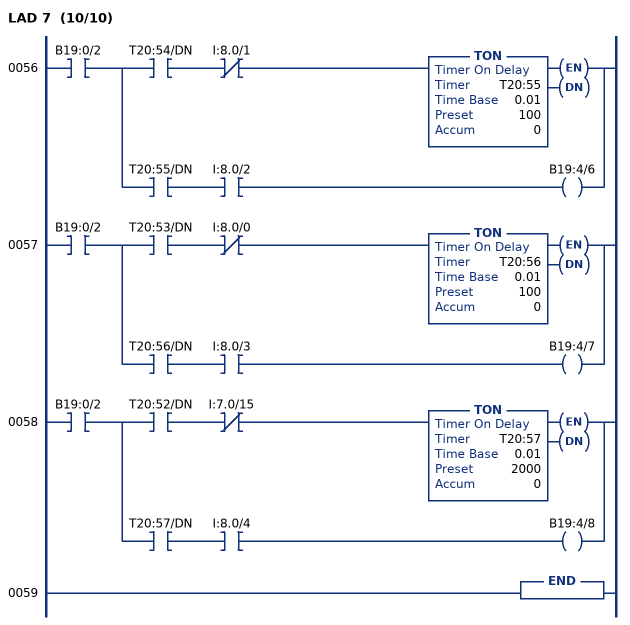
% Rung: 56 %
SOR XIC B19:0/2 BST XIC T20:54/DN XIO I:8.0/1 TON T20:55 0.01 100 0 NXB XIC T20:55/DN XIC I:8.0/2 OTE B19:4/6 BND EOR
% Rung: 57 %
SOR XIC B19:0/2 BST XIC T20:53/DN XIO I:8.0/0 TON T20:56 0.01 100 0 NXB XIC T20:56/DN XIC I:8.0/3 OTE B19:4/7 BND EOR
% Rung: 58 %
SOR XIC B19:0/2 BST XIC T20:52/DN XIO I:7.0/15 TON T20:57 0.01 2000 0 NXB XIC T20:57/DN XIC I:8.0/4 OTE B19:4/8 BND EOR
% Rung: 59 %
SOR END EOR

LADDER 8
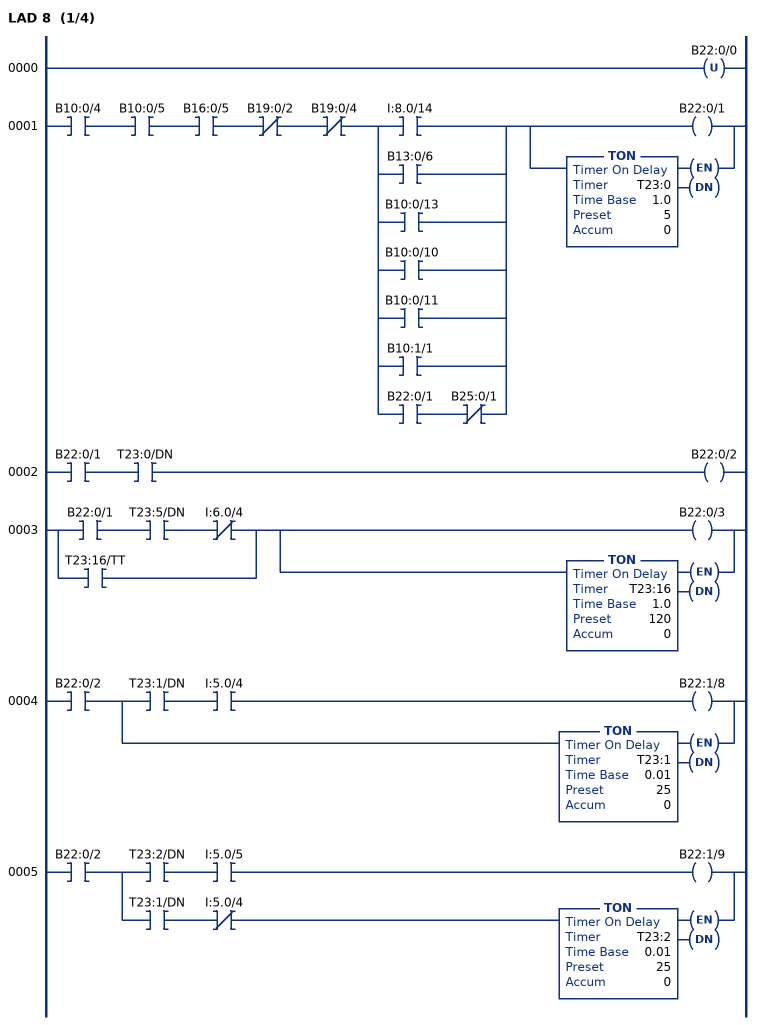
% Rung: 0 %
SOR OTU B22:0/0 EOR
% Rung: 1 %
SOR XIC B10:0/4 XIC B10:0/5 XIC B16:0/5 XIO B19:0/2 XIO B19:0/4 BST XIC I:8.0/14 NXB XIC B13:0/6 NXB XIC B10:0/13 NXB XIC B10:0/10 NXB XIC B10:0/11 NXB XIC B10:1/1 NXB XIC B22:0/1 XIO B25:0/1 BND BST OTE B22:0/1 NXB TON T23:0 1.0 5 0 BND EOR
% Rung: 2 %
SOR XIC B22:0/1 XIC T23:0/DN OTE B22:0/2 EOR
% Rung: 3 %
SOR BST XIC B22:0/1 XIC T23:5/DN XIO I:6.0/4 NXB XIC T23:16/TT BND BST OTE B22:0/3 NXB TON T23:16 1.0 120 0 BND EOR
% Rung: 4 %
SOR XIC B22:0/2 BST XIC T23:1/DN XIC I:5.0/4 OTE B22:1/8 NXB TON T23:1 0.01 25 0 BND EOR
% Rung: 5 %
SOR XIC B22:0/2 BST XIC T23:2/DN XIC I:5.0/5 OTE B22:1/9 NXB XIC T23:1/DN XIO I:5.0/4 TON T23:2 0.01 25 0 BND EOR

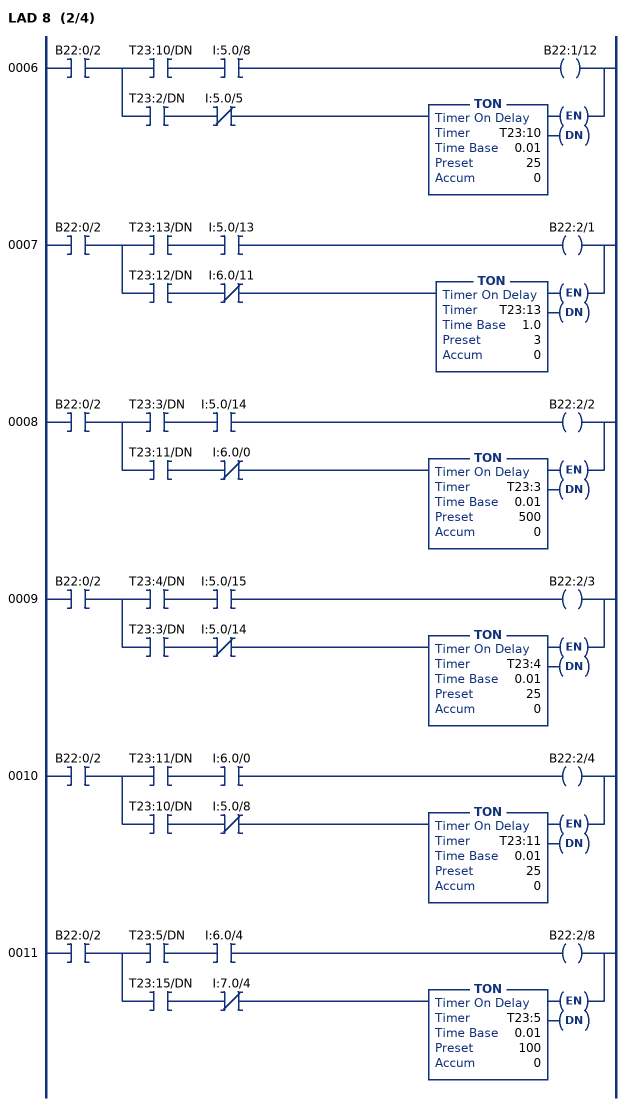
% Rung: 6 %
SOR XIC B22:0/2 BST XIC T23:10/DN XIC I:5.0/8 OTE B22:1/12 NXB XIC T23:2/DN XIO I:5.0/5 TON T23:10 0.01 25 0 BND EOR
% Rung: 7 %
SOR XIC B22:0/2 BST XIC T23:13/DN XIC I:5.0/13 OTE B22:2/1 NXB XIC T23:12/DN XIO I:6.0/11 TON T23:13 1.0 3 0 BND EOR
% Rung: 8 %
SOR XIC B22:0/2 BST XIC T23:3/DN XIC I:5.0/14 OTE B22:2/2 NXB XIC T23:11/DN XIO I:6.0/0 TON T23:3 0.01 500 0 BND EOR
% Rung: 9 %
SOR XIC B22:0/2 BST XIC T23:4/DN XIC I:5.0/15 OTE B22:2/3 NXB XIC T23:3/DN XIO I:5.0/14 TON T23:4 0.01 25 0 BND EOR
% Rung: 10 %
SOR XIC B22:0/2 BST XIC T23:11/DN XIC I:6.0/0 OTE B22:2/4 NXB XIC T23:10/DN XIO I:5.0/8 TON T23:11 0.01 25 0 BND EOR
% Rung: 11 %
SOR XIC B22:0/2 BST XIC T23:5/DN XIC I:6.0/4 OTE B22:2/8 NXB XIC T23:15/DN XIO I:7.0/4 TON T23:5 0.01 100 0 BND EOR

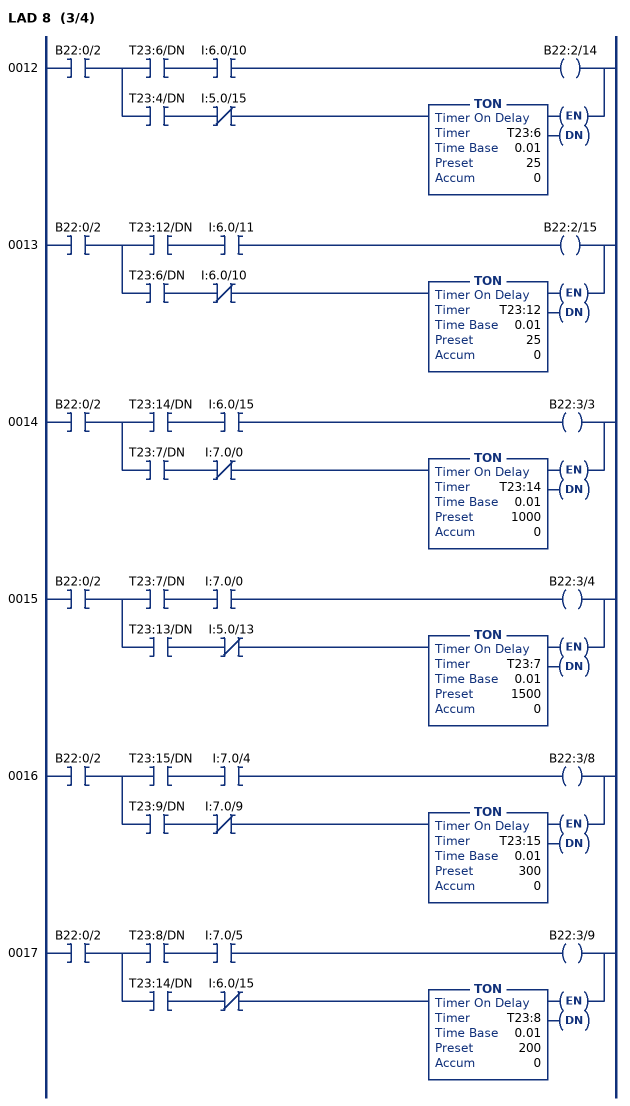
% Rung: 12 %
SOR XIC B22:0/2 BST XIC T23:6/DN XIC I:6.0/10 OTE B22:2/14 NXB XIC T23:4/DN XIO I:5.0/15 TON T23:6 0.01 25 0 BND EOR
% Rung: 13 %
SOR XIC B22:0/2 BST XIC T23:12/DN XIC I:6.0/11 OTE B22:2/15 NXB XIC T23:6/DN XIO I:6.0/10 TON T23:12 0.01 25 0 BND EOR
% Rung: 14 %
SOR XIC B22:0/2 BST XIC T23:14/DN XIC I:6.0/15 OTE B22:3/3 NXB XIC T23:7/DN XIO I:7.0/0 TON T23:14 0.01 1000 0 BND EOR
% Rung: 15 %
SOR XIC B22:0/2 BST XIC T23:7/DN XIC I:7.0/0 OTE B22:3/4 NXB XIC T23:13/DN XIO I:5.0/13 TON T23:7 0.01 1500 0 BND EOR
% Rung: 16 %
SOR XIC B22:0/2 BST XIC T23:15/DN XIC I:7.0/4 OTE B22:3/8 NXB XIC T23:9/DN XIO I:7.0/9 TON T23:15 0.01 300 0 BND EOR
% Rung: 17 %
SOR XIC B22:0/2 BST XIC T23:8/DN XIC I:7.0/5 OTE B22:3/9 NXB XIC T23:14/DN XIO I:6.0/15 TON T23:8 0.01 200 0 BND EOR

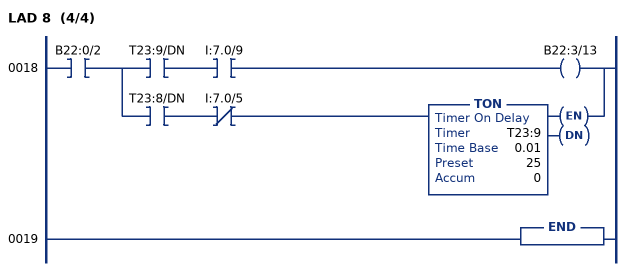
% Rung: 18 %
SOR XIC B22:0/2 BST XIC T23:9/DN XIC I:7.0/9 OTE B22:3/13 NXB XIC T23:8/DN XIO I:7.0/5 TON T23:9 0.01 25 0 BND EOR
% Rung: 19 %
SOR END EOR

LADDER 9
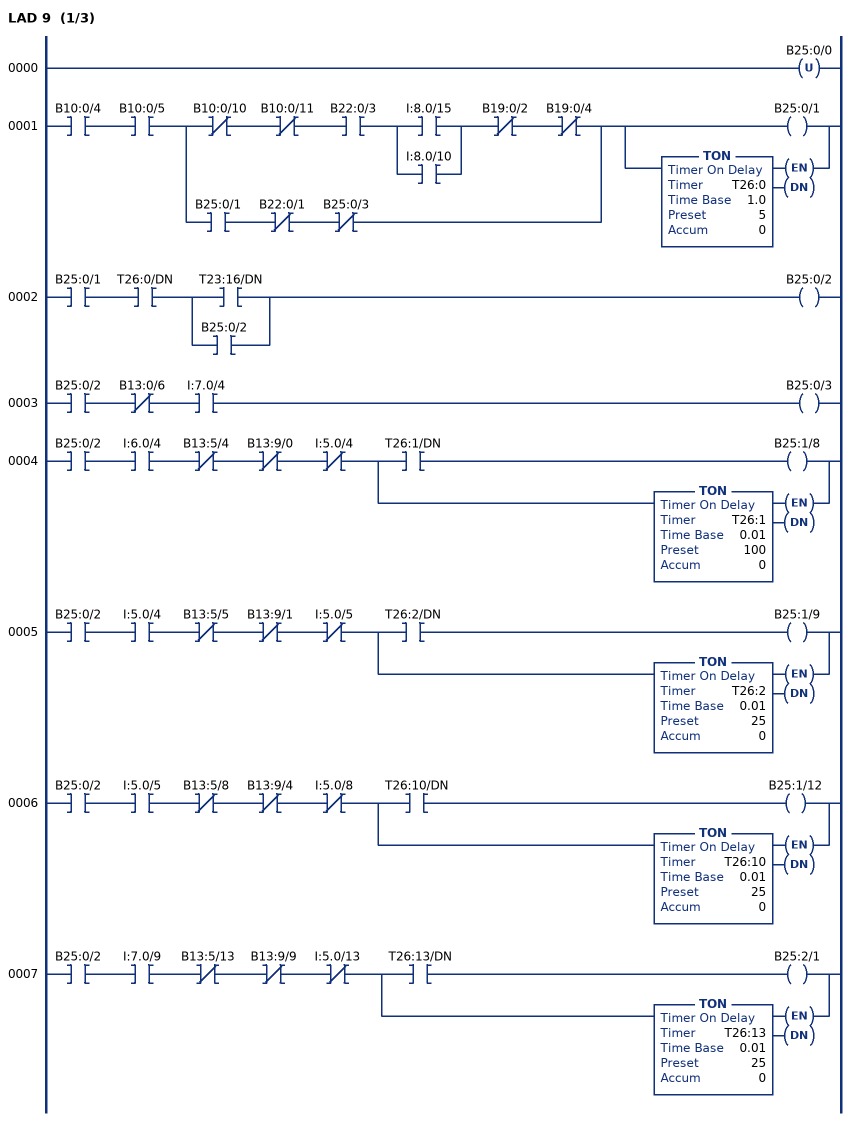
% Rung: 0 %
SOR OTU B25:0/0 EOR
% Rung: 1 %
SOR XIC B10:0/4 XIC B10:0/5 BST XIO B10:0/10 XIO B10:0/11 XIC B22:0/3 BST XIC I:8.0/15 NXB XIC I:8.0/10 BND XIO B19:0/2 XIO B19:0/4 NXB XIC B25:0/1 XIO B22:0/1 XIO B25:0/3 BND BST OTE B25:0/1 NXB TON T26:0 1.0 5 0 BND EOR
% Rung: 2 %
SOR XIC B25:0/1 XIC T26:0/DN BST XIC T23:16/DN NXB XIC B25:0/2 BND OTE B25:0/2 EOR
% Rung: 3 %
SOR XIC B25:0/2 XIO B13:0/6 XIC I:7.0/4 OTE B25:0/3 EOR
% Rung: 4 %
SOR XIC B25:0/2 XIC I:6.0/4 XIO B13:5/4 XIO B13:9/0 XIO I:5.0/4 BST XIC T26:1/DN OTE B25:1/8 NXB TON T26:1 0.01 100 0 BND EOR
% Rung: 5 %
SOR XIC B25:0/2 XIC I:5.0/4 XIO B13:5/5 XIO B13:9/1 XIO I:5.0/5 BST XIC T26:2/DN OTE B25:1/9 NXB TON T26:2 0.01 25 0 BND EOR
% Rung: 6 %
SOR XIC B25:0/2 XIC I:5.0/5 XIO B13:5/8 XIO B13:9/4 XIO I:5.0/8 BST XIC T26:10/DN OTE B25:1/12 NXB TON T26:10 0.01 25 0 BND EOR
% Rung: 7 %
SOR XIC B25:0/2 XIC I:7.0/9 XIO B13:5/13 XIO B13:9/9 XIO I:5.0/13 BST XIC T26:13/DN OTE B25:2/1 NXB TON T26:13 0.01 25 0 BND EOR

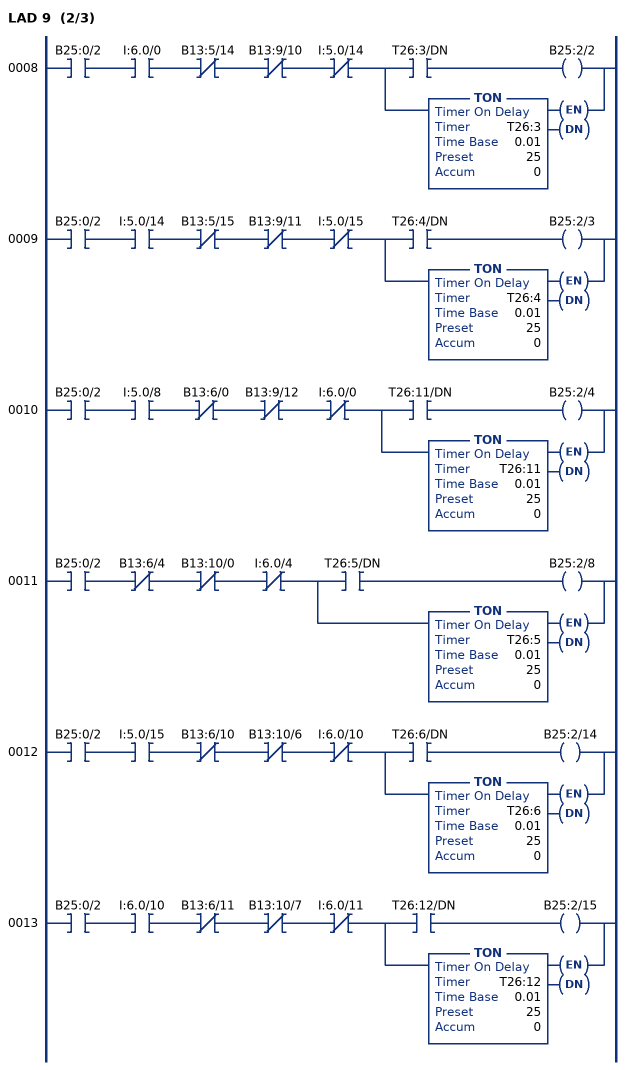
% Rung: 8 %
SOR XIC B25:0/2 XIC I:6.0/0 XIO B13:5/14 XIO B13:9/10 XIO I:5.0/14 BST XIC T26:3/DN OTE B25:2/2 NXB TON T26:3 0.01 25 0 BND EOR
% Rung: 9 %
SOR XIC B25:0/2 XIC I:5.0/14 XIO B13:5/15 XIO B13:9/11 XIO I:5.0/15 BST XIC T26:4/DN OTE B25:2/3 NXB TON T26:4 0.01 25 0 BND EOR
% Rung: 10 %
SOR XIC B25:0/2 XIC I:5.0/8 XIO B13:6/0 XIO B13:9/12 XIO I:6.0/0 BST XIC T26:11/DN OTE B25:2/4 NXB TON T26:11 0.01 25 0 BND EOR
% Rung: 11 %
SOR XIC B25:0/2 XIO B13:6/4 XIO B13:10/0 XIO I:6.0/4 BST XIC T26:5/DN OTE B25:2/8 NXB TON T26:5 0.01 25 0 BND EOR
% Rung: 12 %
SOR XIC B25:0/2 XIC I:5.0/15 XIO B13:6/10 XIO B13:10/6 XIO I:6.0/10 BST XIC T26:6/DN OTE B25:2/14 NXB TON T26:6 0.01 25 0 BND EOR
% Rung: 13 %
SOR XIC B25:0/2 XIC I:6.0/10 XIO B13:6/11 XIO B13:10/7 XIO I:6.0/11 BST XIC T26:12/DN OTE B25:2/15 NXB TON T26:12 0.01 25 0 BND EOR

